{attribute 'qualified_only'}
VAR_GLOBAL
	stXAxis :AXIS_REF;
	stXaxisStatus : ST_AxisStatus;
	
END_VAR

(* stored: Version 1.1.0.1, ProductVersion 3.1.4024.3
   GVL GVL_NC: Id {4af7a3fe-5e71-4c16-a01b-bc4bf8fbd493} *)
